// TIA Portal project "Sorting_Station" (V17)

(* hardware
DEVICE "S7-1200 station_1"  S7-1200 Station
   slot 0: "Rack_0"  S7-1200 Rack  Rack  V1.0
   slot 1: "PLC_1"  CPU 1214C DC/DC/DC  6ES7 214-1AG40-0XB0  V4.5
   slot 2: "DI 8/DQ 8x24VDC_1"  SM 1223 DI8/DQ8 x 24VDC  6ES7 223-1BH30-0XB0  V1.0
   slot 3: "AQ 2x14BIT_1"  SM 1232 AQ2  6ES7 232-4HB32-0XB0  V2.1
DEVICE "HMI_1"  KTP700 Basic PN
   slot 0: "HMI_1"  KTP700 Basic PN  6AV2 123-2GB03-0AX0  17.0.0.0
   slot 1: "HMI_RT_1"  KTP700 Basic PN  6AV2 123-2GB03-0AX0  17.0.0.0
   slot 5: "HMI_1.IE_CP_1"  PROFINET Interface  17.0.0.0
      slot 1: "PROFINET Interface_1"  PROFINET Interface
         slot 1: "Port_1"  Port
*)

// ===== PLC "PLC_1"  CPU 1214C DC/DC/DC =====

VAR_GLOBAL   // PLC tag table "Default tag table"
   "Memory_StartPB_HMI" AT %M0.0 : Bool;
END_VAR

VAR_GLOBAL   // PLC tag table "Tag_table_sorting_station"
   "I -A1" AT %I0.0 : Bool;   // Return signal E-Stop OK
   "I -K0" AT %I0.1 : Bool;   // main switch ON
   "I -S1" AT %I0.3 : Bool;   // PB Auto start
   "I -S2" AT %I0.4 : Bool;   // PB Auto Stop(in initial state)
   "I -B1" AT %I0.5 : Bool;   // Sensor cylinder M4 Retracted
   "I -B2" AT %I0.6 : Bool;   // Sensor Cylinder M4 Extented
   "I -B3" AT %I0.7 : Bool;   // Sensor motor M1 Active
   "I -B4" AT %I1.0 : Bool;   // Sensor at chute Occupied
   "I -B5" AT %I1.1 : Bool;   // Sensor metal part
   "I -B6" AT %I1.2 : Bool;   // Sensor part in front of cylinder M4
   "I -B7" AT %I1.3 : Bool;   // Sensor at End of conveyor
   "I -S3" AT %I1.4 : Bool;   // PB conveyor manual mode-Forward
   "I -S4" AT %I1.5 : Bool;   // PB conveyor manual mode-Reverse
   "I -S5" AT %I1.6 : Bool;   // PB manaul mode cylinder M4 retracts
   "I -S6" AT %I1.7 : Bool;   // PB manual mode cylinder M4 extends
   "I -S0" AT %I0.2 : Bool;   // mode selector- manual(0)/Auto(1)
   "Q -Q1" AT %Q0.0 : Bool;   // Conveyor motor M1 forward - fix speed
   "Q -Q2" AT %Q0.1 : Bool;   // Conveyor motor M1 reverse - fix speed
   "Q -Q3" AT %Q0.2 : Bool;   // Conveyor motor M1 - Variable Speed
   "Q -M2" AT %Q0.3 : Bool;   // Cylinder M4 retracts
   "Q -M3" AT %Q0.4 : Bool;   // Cylinder M4 extends
   "Q -P1" AT %Q0.5 : Bool;   // Display- main switch ON
   "Q -P2" AT %Q0.6 : Bool;   // Display- Manual mode
   "Q -P3" AT %Q0.7 : Bool;   // Display- auto mode
   "Q -P4" AT %Q1.0 : Bool;   // Display- Emergency stop activated
   "Q -P5" AT %Q1.1 : Bool;   // Display- Auto mode started
   "Q -P6" AT %Q1.2 : Bool;   // Display- Cylinder M4 Retracted
   "Q -P7" AT %Q1.3 : Bool;   // Display- Cylinder M4 Extended
   "AI -B8" AT %IW64 : Word;   // Sensor Actual value speed of motor +\- 10V
   "AI -B9" AT %IW66 : Word;   // Set point Specification via Potentiometer +\-10V
   "AO -U1" AT %QW64 : Word;   // Manipulated value speed of motor in 2 direction +\-10V
   "Temp-store-speed" AT %MW25 : Word;   // used to store 16 bit value
END_VAR

DATA_BLOCK "Motor_Auto"   // DB1
{ S7_Optimized_Access := 'FALSE' }
VERSION : 0.1
// stored: InstanceOfName Motor_Auto_mode
"Motor_Auto_mode"
BEGIN
   Setpoint_plastic_count := 5;
END_DATA_BLOCK

DATA_BLOCK "SPEED_MOTOR"   // DB2
{ S7_Optimized_Access := 'TRUE' }
VERSION : 0.1
   VAR
      Speed_Setpoint_Auto : Real := 15.0;
      Speed_Actual_Value : Real := 15.0;
      Positive_Speed : Struct   // Parameters for error/ warning positive speed
         Threshold_error : Real := 15.0;   // Speed Limit / if exceeded an error is displayed
         Threshold_Warning : Real := 10.0;   // Speed Limit / if exceeded an warning is displayed
         Error : Bool := FALSE;   // Error limit exceeded
         Warning : Bool := TRUE;   // Warning limit exceeded
      END_STRUCT;
      Negative_Speed : Struct
         Threshold_error : Real := -16.0;   // Speed Limit / if exceeded an error is displayed
         Threshold_Warning : Real := -10.0;   // Speed Limit / if exceeded an warning is displayed
         Error : Bool := FALSE;   // Error limit exceeded
         Warning : Bool := FALSE;   // Warning limit exceeded
      END_STRUCT;
      speed_setpoint_manual : Real := 5.0;
   END_VAR
BEGIN
END_DATA_BLOCK

DATA_BLOCK "MAGAZINE_PLASTIC"   // DB3
{ S7_Optimized_Access := 'TRUE' }
VERSION : 0.1
   VAR
      Setpoint_plastic_count : Int := 5;
      Actual_plastic_count : Int;
      Reset_plastic_count : Bool;
   END_VAR
BEGIN
END_DATA_BLOCK

DATA_BLOCK "OPERATING_HMI"   // DB4
{ S7_Optimized_Access := 'TRUE' }
VERSION : 0.1
   VAR
      mode_selector : Bool := false;
      automatic_start : Bool;
      automatic_stop : Bool := true;
      reset_counter_plastic : Bool;
      "Alarm Group signals01" : Word;
      "Alarm Ack Group Signals01" : Word;
   END_VAR
BEGIN
END_DATA_BLOCK

FUNCTION_BLOCK "Motor_Auto_mode"   // FB1, FBD
{ S7_Optimized_Access := 'FALSE' }
VERSION : 0.1
// The Memory_automatic_start_stop is latched with Start but only if the reset conditions are not
//  present.
//  
//  The Memory_automatic_start_stop is reset if Stop is present or safety shutoff is active or
//  automatic mode is not activated (manual mode).
//  The Conveyor_motor_automatic_mode output is activated when Memory_automatic_start_stop is
//  set, the enable conditions are met and Memory_conveyor_start_stop is set.
//  To save energy, the conveyor should only run when a part is present.
//  For this reason, the Memory_conveyor_start_stop is set when Sensor_chute_occupied signals a
//  part and reset when Sensor_end_of_conveyor produces a negative edge or safety shutoff is
//  active or automatic mode is not activated (manual mode).
// 
//  Because the Sensor_end_of_conveyor is not able to be mounted directly at the end of the
//  conveyor, the Sensor_end_of_conveyor signal must be stretched.
//  To achieve this, a latching pulse will be inserted between Sensor_end_of_conveyor and the
//  negative edge detection.
   VAR_INPUT
      Automatic_mode_active : Bool;   // Automatic mode activated
      Start : Bool;   // Pushbutton Auto start
      Stop : Bool;   // Pushbutton Auto Stop
      Enable_ok : Bool;   // All enable condition OK
      Sensor_chute_occupied : Bool;   // Sensor at chute occupied
      Safety_shutoff_active : Bool;   // Safety shutoff active e.g. Estop
      Sensor_EndofConveyor : Bool;   // Sensor part at end of conveyor
      Setpoint_plastic_count : Int;
      Reset_Counter_Workpieces_Plastic : Bool;
   END_VAR
   VAR_OUTPUT
      Conveyor_motor_auto_mode : Bool;   // Control of Conveyor motor in Auto mode
      Actual_plastic_count : Int;
   END_VAR
   VAR
      Memory_Automatic_Start_Stop : Bool;   // Memory used for start/stop automatic mode
      Memory_conveyor_start_stop : Bool;
      Memory_Edge_detection : Bool;
      IEC_Timer_Overrun : TP_TIME;
      IEC_Counter_Overrun : CTU_INT;
   END_VAR
   VAR_TEMP   // added for the SCL form of the ladder/FBD networks
      _w1 : Bool;
   END_VAR
BEGIN

REGION Network 1: Counting plastic pieces
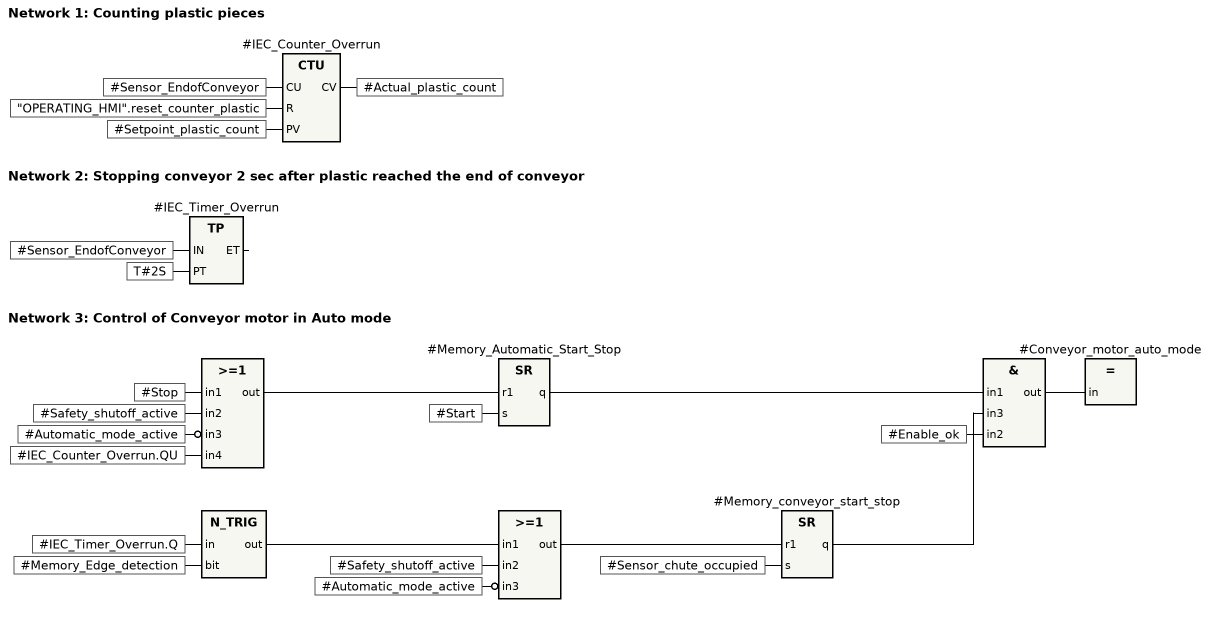
   #IEC_Counter_Overrun(CU := #Sensor_EndofConveyor,   // CTU
                        R := "OPERATING_HMI".reset_counter_plastic,
                        PV := #Setpoint_plastic_count,
                        CV => #Actual_plastic_count);
END_REGION

REGION Network 2: Stopping conveyor 2 sec after plastic reached the end of conveyor
   #IEC_Timer_Overrun(IN := #Sensor_EndofConveyor, PT := T#2S);   // TP
END_REGION

REGION Network 3: Control of Conveyor motor in Auto mode
   IF #Start THEN
       #Memory_Automatic_Start_Stop := TRUE;   // SR flip-flop
   END_IF;
   IF #Stop OR #Safety_shutoff_active OR NOT #Automatic_mode_active OR #IEC_Counter_Overrun.QU THEN
       #Memory_Automatic_Start_Stop := FALSE;
   END_IF;
   #_w1 := NOT #IEC_Timer_Overrun.Q AND #Memory_Edge_detection;   // falling edge
   #Memory_Edge_detection := #IEC_Timer_Overrun.Q;
   IF #Sensor_chute_occupied THEN
       #Memory_conveyor_start_stop := TRUE;   // SR flip-flop
   END_IF;
   IF #_w1 OR #Safety_shutoff_active OR NOT #Automatic_mode_active THEN
       #Memory_conveyor_start_stop := FALSE;
   END_IF;
   #Conveyor_motor_auto_mode := #Memory_Automatic_Start_Stop AND #Memory_conveyor_start_stop AND #Enable_ok;
END_REGION
END_FUNCTION_BLOCK

FUNCTION "Motor_manual_Mode" : Void   // FC1, FBD
TITLE = Motor control in manual mode
{ S7_Optimized_Access := 'TRUE' }
VERSION : 0.1
// conveyor motor in manual mode: If the pushbutton_manual_mode is opeerated, the enable conditions are granted and the safety shutoff is not activated the output
// Conveyor_motor_manual_mode is activated.
   VAR_INPUT
      Manual_mode_active : Bool;   // Manual mode activated
      Pushbutton_manual_mode : Bool;   // Pushbutton manual mode conveyor on
      Enable_OK : Bool;   // All enable conditions OK
      Safety_shutoff_active : Bool;   // Saftey shutoff active
      Forward_signal : Bool;   // signal for operation in forward direction
      Backward_signal : Bool;   // signal for operation in reverse direction
      manual_motor_speed : Real;   // speed of motor for manual mode in either direction
   END_VAR
   VAR_OUTPUT
      Conveyor_mode_manual_mode : Bool;   // Control of the conveyor motor in manual mode
      Output_motor_speed : Real;   // speed of motor in manual mode
   END_VAR
   VAR_TEMP
      negative_value : Real;
      "Speed*2" : Real;
   END_VAR
BEGIN

REGION Network 1: Control of the conveyor in manual mode.
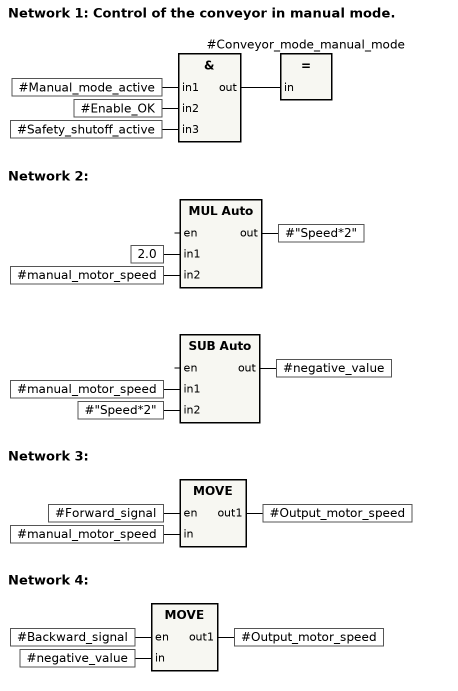
   #Conveyor_mode_manual_mode := #Manual_mode_active AND #Enable_OK AND #Safety_shutoff_active;
END_REGION

REGION Network 2
   #"Speed*2" := 2.0 * #manual_motor_speed;
   #negative_value := #manual_motor_speed - #"Speed*2";
END_REGION

REGION Network 3
   IF #Forward_signal THEN #Output_motor_speed := #manual_motor_speed; END_IF;
END_REGION

REGION Network 4
   IF #Backward_signal THEN #Output_motor_speed := #negative_value; END_IF;
END_REGION
END_FUNCTION

FUNCTION "Copy 16bit data" : Void   // FC2, SCL
{ S7_Optimized_Access := 'TRUE' }
VERSION : 0.1
   VAR_INPUT
      "Copy speed from" : Int;
   END_VAR
   VAR_OUTPUT
      "Copy speed to" : Int;
   END_VAR
BEGIN
   #"Copy speed to" := #"Copy speed from";
END_FUNCTION

FUNCTION "Assign_discrete_alarms" : Void   // FC3, FBD
{ S7_Optimized_Access := 'TRUE' }
VERSION : 0.1
   VAR_INPUT
      discrete_alarm_X0 : Bool;
      discrete_alarm_X1 : Bool;
      discrete_alarm_X2 : Bool;
      discrete_alarm_X3 : Bool;
   END_VAR
   VAR_OUTPUT
      group_signal01 : Word;
   END_VAR
BEGIN

REGION Network 1
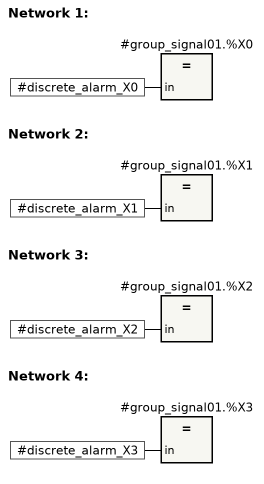
   #group_signal01.%X0 := #discrete_alarm_X0;
END_REGION

REGION Network 2
   #group_signal01.%X1 := #discrete_alarm_X1;
END_REGION

REGION Network 3
   #group_signal01.%X2 := #discrete_alarm_X2;
END_REGION

REGION Network 4
   #group_signal01.%X3 := #discrete_alarm_X3;
END_REGION
END_FUNCTION

FUNCTION "MOTOR_SPEEDMONITORING" : Void   // FC11, FBD
{ S7_Optimized_Access := 'TRUE' }
VERSION : 0.1
// In the "MOTOR_SPEED_MONITORING" [FC11] function, the actual value is made available at 
// B8 as an analog value and is queried at an input of the "MOTOR_SPEEDMONITORING" [FC11]
//  function.
//  The actual speed value is scaled to revolutions per minute (range: +/- 50 rpm) and made
//  available at an output.
//  The following four limits can be specified at the block inputs in order to monitor them in the
//  function:
//  Speed > Speed limit error max
//  Speed > Speed limit warning max
//  Speed  < Speed limit warning min
//  Speed  < Speed limit warning min
//  If a limit is exceeded or undershot, the value TRUE (1) is assigned to the corresponding output
//  bit.
//  If a fault is present, the safety shutoff of the "MOTOR_AUTO" [FB1] function block is to be
//  triggered
   VAR_INPUT
      Actual_Speed_AI : Int;
      Speed_limit_error_max : Real;
      Speed_limit_warning_max : Real;
      Speed_limit_warning_min : Real;
      Speed_limit_error_min : Real;
   END_VAR
   VAR_OUTPUT
      Speed_warning_max : Bool;
      Speed_warning_min : Bool;
      Speed_error_max : Bool;
      Speed_error_min : Bool;
      Motor_speed_AO : Real;
   END_VAR
   VAR_TEMP
      Motor_speed_Norm : Real;
      Actual_speed_Scaled : Real;
   END_VAR
BEGIN

REGION Network 1: Normalisation
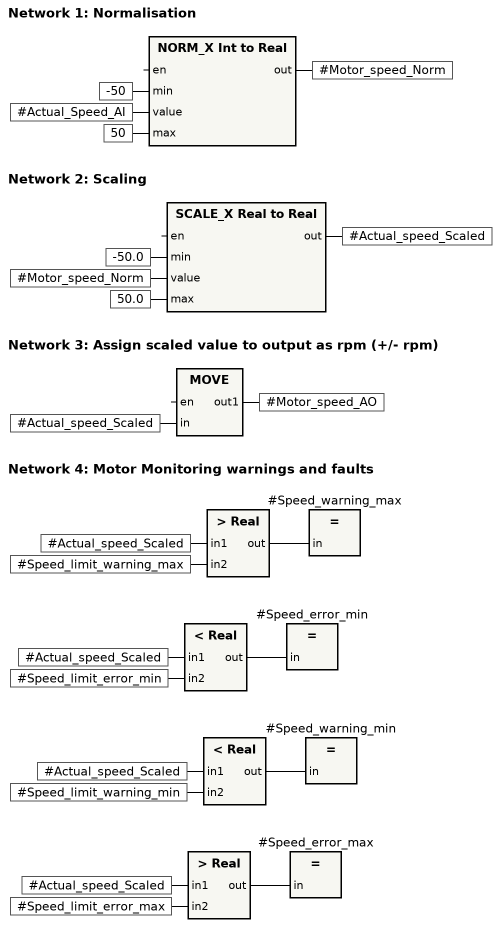
   #Motor_speed_Norm := NORM_X(MIN := -50, VALUE := #Actual_Speed_AI, MAX := 50);
END_REGION

REGION Network 2: Scaling
   #Actual_speed_Scaled := SCALE_X(MIN := -50.0, VALUE := #Motor_speed_Norm, MAX := 50.0);
END_REGION

REGION Network 3: Assign scaled value to output as rpm (+/- rpm)
   #Motor_speed_AO := #Actual_speed_Scaled;
END_REGION

REGION Network 4: Motor Monitoring warnings and faults
   #Speed_warning_max := #Actual_speed_Scaled > #Speed_limit_warning_max;
   #Speed_error_min := #Actual_speed_Scaled < #Speed_limit_error_min;
   #Speed_warning_min := #Actual_speed_Scaled < #Speed_limit_warning_min;
   #Speed_error_max := #Actual_speed_Scaled > #Speed_limit_error_max;
END_REGION
END_FUNCTION

ORGANIZATION_BLOCK "Main"   // OB1, FBD, ProgramCycle
TITLE = "Main Program Sweep (Cycle)"
{ S7_Optimized_Access := 'TRUE' }
VERSION : 0.1
// The "MOTOR_AUTO" [FB1] function block controls a conveyor in automatic mode.
//  The Memory_Automatic_Start_Stop is switched on in a latching manner with Start, but only if the
//  reset conditions are not present.
//  The Memory_Automatic_Start_Stop is to be reset if Stop is pending, the safety shutoff is active
//  or automatic mode is not activated from the visualization.
//  The Automatic_Motor output is controlled when Memory_Automatic_Start_Stop is set, the
//  enabling conditions are met and Memory_Conveyor_Start_Stop is set.
//  For energy saving reasons, the conveyor is to run only when a transport part is present.
//  Therefore, Memory_Conveyor_Start_Stop is set if Sensor_slide signals a part and is reset if
//  Sensor_end_of_conveyor generates a negative edge or the safety shutoff is active or automatic
//  mode is not activated (manual mode).
//  Because Sensor_end_of_conveyor is not mounted directly at the end of the conveyor, a signal
//  delay of the Sensor_end_of_conveyor signal is programmed.
//  The magazine for plastics holds only five parts. Therefore, the parts are counted at the end of
//  the conveyor. If the magazine contains five parts, automatic mode is to be stopped. After the
//  magazine is emptied, automatic mode is restarted with another Start, once the counter has been
//  reset from the visualization.
//  The speed is specified with an input in the "MOTOR_SPEEDCONTROL" [FC10] function in
//  revolutions per minute (range: +/- 50 rpm).
//  The speed setpoint is first checked in the function for correct input in the range +/- 50 rpm.
//  If the speed setpoint is outside the range +/- 50 rpm, the value 0 is output at the speed setpoint
//  output. The value TRUE (1) is assigned to the return value of the function (Ret_Val).
//  If the specified speed is in the range +/- 50 rpm, this value is first scaled to the range 0…1 and
//  then scaled for the output as manipulated speed value at the analog output to +/- 27648 with
//  data type 16-bit integer (Int).
//  In the "MOTOR_SPEED_MONITORING" [FC11] function, the actual value is made available at 
// B8 as an analog value and is queried at an input of the "MOTOR_SPEEDMONITORING" [FC11]
//  function.
//  The actual speed value is scaled to revolutions per minute (range: +/- 50 rpm) and made
//  available at an output.
//  The following four limits can be specified at the block inputs in order to monitor them in the
//  function:
//  Speed > Speed limit error max
//  Speed > Speed limit warning max
//  Speed  < Speed limit warning min
//  Speed  < Speed limit warning min
//  If a limit is exceeded or undershot, the value TRUE (1) is assigned to the corresponding output
//  bit.
//  If a fault is present, the safety shutoff of the "MOTOR_AUTO" [FB1] function block is to be
//  triggered.
//  Speed setpoint and actual speed value as well as the positive and negative error and warning
//  limits are created in the "SPEED_MOTOR" [DB2] data block, as are the error and warning bits.
//  The setpoint and actual value of the counter for plastic parts will be specified and displayed in
//  the global "MAGAZINE_PLASTIC" [DB3] data block. These values are connected with the
//  "MOTOR_AUTO" [FB1] function block via an input for specification of the setpoint and via an
//  output for display of the actual value
   VAR_INPUT
      Initial_Call : Bool;   // Initial call of this OB
      Remanence : Bool;   // =True, if remanent data are available
   END_VAR
BEGIN

REGION Network 1: Delete this block if you have real motor connected and actual feedback from field
   // Modify MW25 to read Motor speed value in HMI
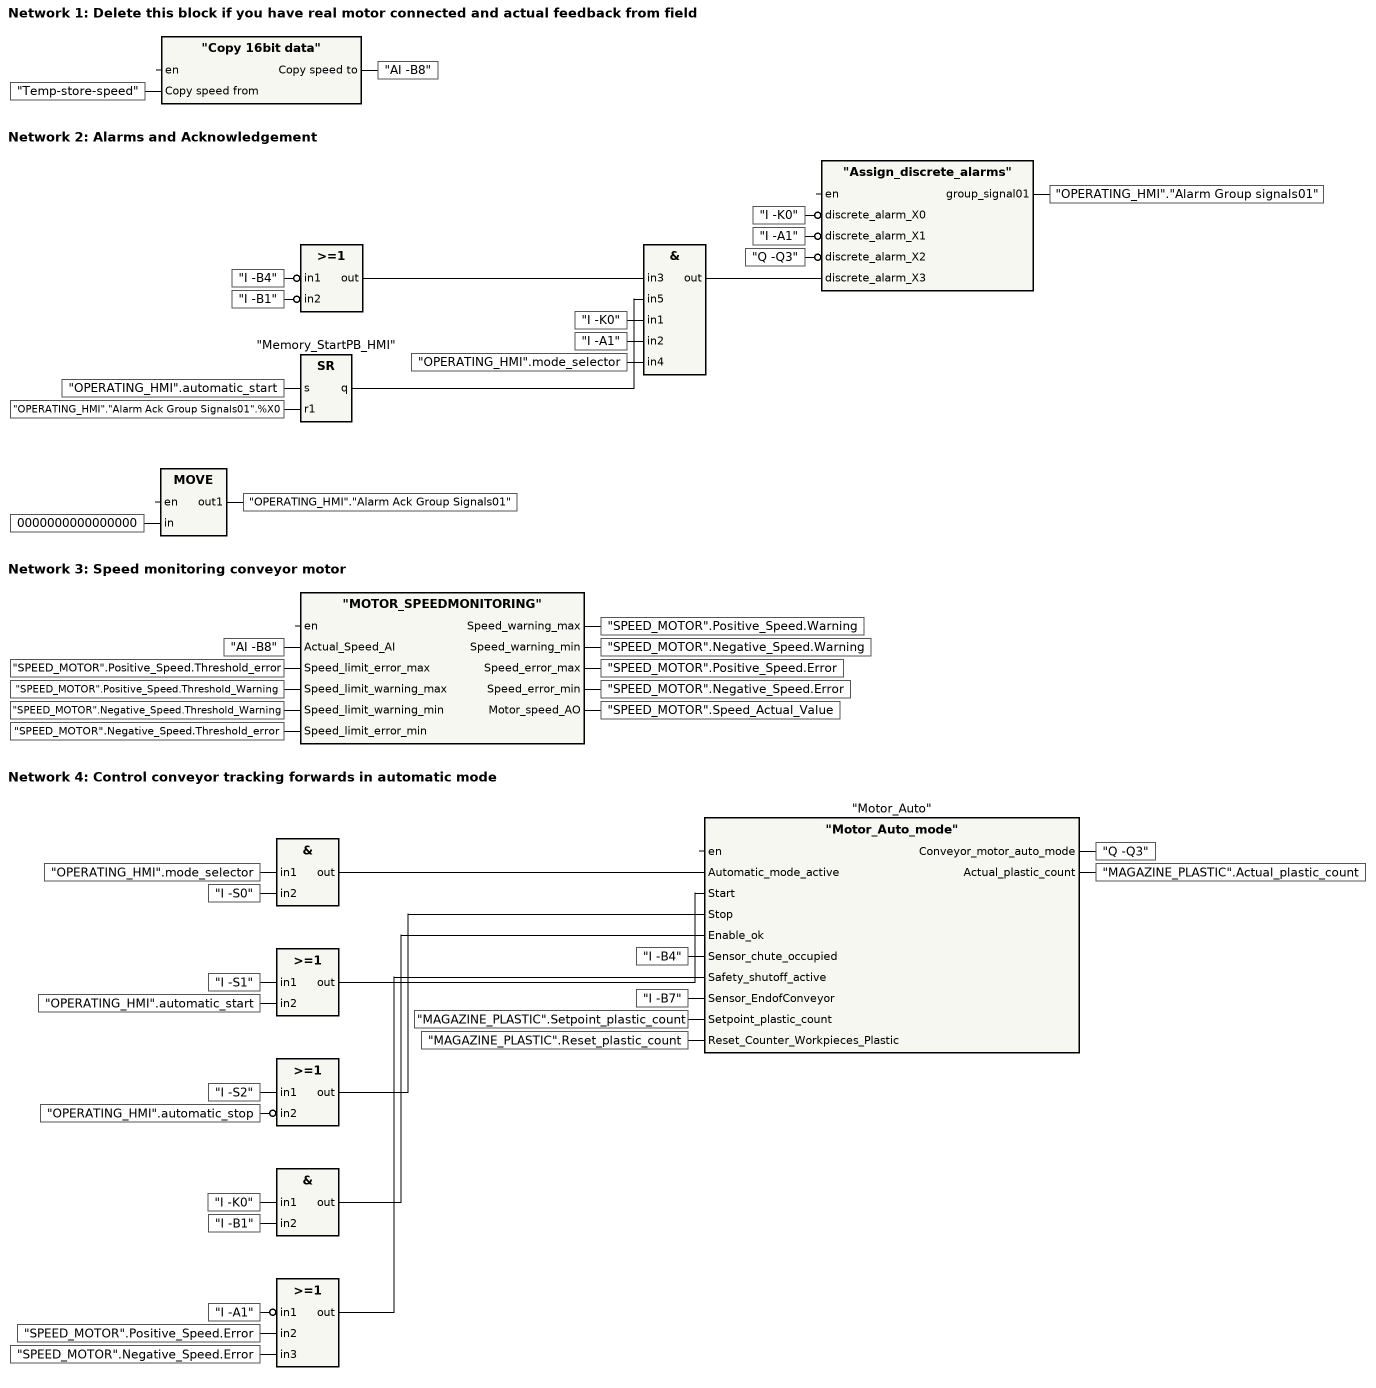
   "Copy 16bit data"("Copy speed from" := "Temp-store-speed", "Copy speed to" => "AI -B8");
END_REGION

REGION Network 2: Alarms and Acknowledgement
   IF "OPERATING_HMI".automatic_start THEN
       "Memory_StartPB_HMI" := TRUE;   // SR flip-flop
   END_IF;
   IF "OPERATING_HMI"."Alarm Ack Group Signals01".%X0 THEN "Memory_StartPB_HMI" := FALSE; END_IF;
   "Assign_discrete_alarms"(discrete_alarm_X0 := NOT "I -K0",
                           discrete_alarm_X1 := NOT "I -A1",
                           discrete_alarm_X2 := NOT "Q -Q3",
                           discrete_alarm_X3 := (NOT "I -B4" OR NOT "I -B1") AND "Memory_StartPB_HMI" AND "I -K0" AND "I -A1" AND "OPERATING_HMI".mode_selector,
                           group_signal01 => "OPERATING_HMI"."Alarm Group signals01");
   "OPERATING_HMI"."Alarm Ack Group Signals01" := 0000000000000000;
END_REGION

REGION Network 3: Speed monitoring conveyor motor
   "MOTOR_SPEEDMONITORING"(Actual_Speed_AI := "AI -B8",
                           Speed_limit_error_max := "SPEED_MOTOR".Positive_Speed.Threshold_error,
                           Speed_limit_warning_max := "SPEED_MOTOR".Positive_Speed.Threshold_Warning,
                           Speed_limit_warning_min := "SPEED_MOTOR".Negative_Speed.Threshold_Warning,
                           Speed_limit_error_min := "SPEED_MOTOR".Negative_Speed.Threshold_error,
                           Speed_warning_max => "SPEED_MOTOR".Positive_Speed.Warning,
                           Speed_warning_min => "SPEED_MOTOR".Negative_Speed.Warning,
                           Speed_error_max => "SPEED_MOTOR".Positive_Speed.Error,
                           Speed_error_min => "SPEED_MOTOR".Negative_Speed.Error,
                           Motor_speed_AO => "SPEED_MOTOR".Speed_Actual_Value);
END_REGION

REGION Network 4: Control conveyor tracking forwards in automatic mode
   "Motor_Auto"(Automatic_mode_active := "OPERATING_HMI".mode_selector AND "I -S0",   // "Motor_Auto_mode"
                Start := "I -S1" OR "OPERATING_HMI".automatic_start,
                Stop := "I -S2" OR NOT "OPERATING_HMI".automatic_stop,
                Enable_ok := "I -K0" AND "I -B1",
                Sensor_chute_occupied := "I -B4",
                Safety_shutoff_active := NOT "I -A1" OR "SPEED_MOTOR".Positive_Speed.Error OR "SPEED_MOTOR".Negative_Speed.Error,
                Sensor_EndofConveyor := "I -B7",
                Setpoint_plastic_count := "MAGAZINE_PLASTIC".Setpoint_plastic_count,
                Reset_Counter_Workpieces_Plastic := "MAGAZINE_PLASTIC".Reset_plastic_count,
                Conveyor_motor_auto_mode => "Q -Q3",
                Actual_plastic_count => "MAGAZINE_PLASTIC".Actual_plastic_count);
END_REGION

REGION Network 5: Control conveyor motor forwards in manual mode
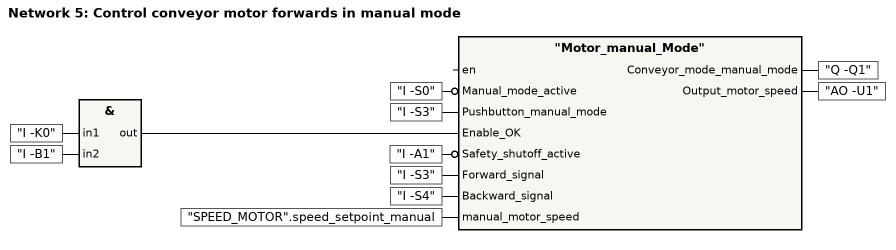
   "Motor_manual_Mode"(Manual_mode_active := NOT "I -S0",
                       Pushbutton_manual_mode := "I -S3",
                       Enable_OK := "I -K0" AND "I -B1",
                       Safety_shutoff_active := NOT "I -A1",
                       Forward_signal := "I -S3",
                       Backward_signal := "I -S4",
                       manual_motor_speed := "SPEED_MOTOR".speed_setpoint_manual,
                       Conveyor_mode_manual_mode => "Q -Q1",
                       Output_motor_speed => "AO -U1");
END_REGION
END_ORGANIZATION_BLOCK

ORGANIZATION_BLOCK "Cyclic interrupt"   // OB30, FBD, CyclicInterrupt
{ S7_Optimized_Access := 'TRUE' }
VERSION : 0.1
   VAR_INPUT
      Initial_Call : Bool;   // Initial call of this OB
      Event_Count : Int;   // Events discarded
   END_VAR
BEGIN

REGION Network 1
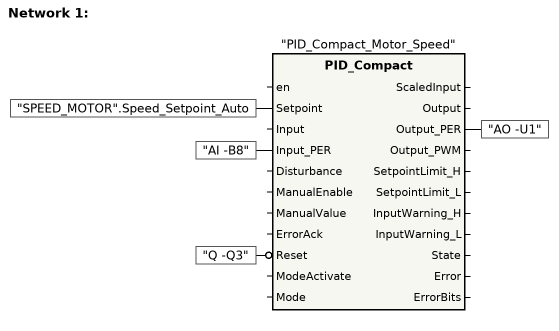
   "PID_Compact_Motor_Speed"(Setpoint := "SPEED_MOTOR".Speed_Setpoint_Auto,   // PID_Compact
                           Input_PER := "AI -B8",
                           Reset := NOT "Q -Q3",
                           Output_PER => "AO -U1");
END_REGION
END_ORGANIZATION_BLOCK

(* ===== HMI "HMI_RT_1" =====
system functions are stored by id; their names below are inferred from use
connection "HMI_Connection_1": ETHERNET, SMART_S7_1200_OMS

HMI tags "Default tag table"
   "Tag_ScreenNumber" : UInt, internal
   "SPEED_MOTOR_Speed_Actual_Value" : Real = PLC SPEED_MOTOR.Speed_Actual_Value, 100 ms
   "I -B4" : Bool = PLC "I -B4" AT %I1.0, 100 ms
   "I -B5" : Bool = PLC "I -B5" AT %I1.1, 100 ms
   "I -B6" : Bool = PLC "I -B6" AT %I1.2, 100 ms
   "I -B7" : Bool = PLC "I -B7" AT %I1.3, 100 ms
   "I -B2" : Bool = PLC "I -B2" AT %I0.6, 100 ms
   "I -B1" : Bool = PLC "I -B1" AT %I0.5, 100 ms
   "I -B3" : Bool = PLC "I -B3" AT %I0.7, 100 ms
   "Q -Q3" : Bool = PLC "Q -Q3" AT %Q0.2, 100 ms
   "OPERATING_HMI_reset_counter_plastic" : Bool = PLC OPERATING_HMI.reset_counter_plastic, 100 ms
   "MAGAZINE_PLASTIC_Actual_plastic_count" : Int = PLC MAGAZINE_PLASTIC.Actual_plastic_count, 100 ms
   "OPERATING_HMI_automatic_start" : Bool = PLC OPERATING_HMI.automatic_start, 100 ms
   "OPERATING_HMI_automatic_stop" : Bool = PLC OPERATING_HMI.automatic_stop, 100 ms
   "I -A1" : Bool = PLC "I -A1" AT %I0.0, 100 ms
   "I -K0" : Bool = PLC "I -K0" AT %I0.1, 100 ms
   "Motor_Auto_Memory_Automatic_Start_Stop" : Bool = PLC Motor_Auto.Memory_Automatic_Start_Stop AT %DB1.DBX10.0, 100 ms
   "SPEED_MOTOR_Speed_Setpoint" : Real = PLC SPEED_MOTOR.Speed_Setpoint_Auto, 100 ms
   "SPEED_MOTOR_Positive_Speed_Threshold_error" : Real = PLC SPEED_MOTOR.Positive_Speed.Threshold_error, 100 ms
   "SPEED_MOTOR_Positive_Speed_Threshold_Warning" : Real = PLC SPEED_MOTOR.Positive_Speed.Threshold_Warning, 100 ms
   "SPEED_MOTOR_Negative_Speed_Threshold_error" : Real = PLC SPEED_MOTOR.Negative_Speed.Threshold_error, 100 ms
   "SPEED_MOTOR_Negative_Speed_Threshold_Warning" : Real = PLC SPEED_MOTOR.Negative_Speed.Threshold_Warning, 100 ms
   "OPERATING_HMI_Group signals01" : Word = PLC OPERATING_HMI."Alarm Group signals01", 1 s
   "MAGAZINE_PLASTIC_Setpoint_plastic_count" : Int = PLC MAGAZINE_PLASTIC.Setpoint_plastic_count, 1 s
   "SPEED_MOTOR_Positive_Speed_Error" : Bool = PLC SPEED_MOTOR.Positive_Speed.Error, 1 s
   "SPEED_MOTOR_Positive_Speed_Warning" : Bool = PLC SPEED_MOTOR.Positive_Speed.Warning, 1 s
   "SPEED_MOTOR_Negative_Speed_Warning" : Bool = PLC SPEED_MOTOR.Negative_Speed.Warning, 1 s
   "SPEED_MOTOR_Negative_Speed_Error" : Bool = PLC SPEED_MOTOR.Negative_Speed.Error, 1 s
   "Motor_Auto_Setpoint_plastic_count" : Int = PLC Motor_Auto.Setpoint_plastic_count AT %DB1.DBW2, 1 s
   "OPERATING_HMI_mode_selector" : Bool = PLC OPERATING_HMI.mode_selector, 1 s
   "SPEED_MOTOR_speed_setpoint_manual" : Real = PLC SPEED_MOTOR.speed_setpoint_manual, 1 s
   "OPERATING_HMI_Alarm Ack Group Signals01" : Word = PLC OPERATING_HMI."Alarm Ack Group Signals01", 1 s

discrete alarms
   1: 'Main switch OFF', class Warnings, trigger "OPERATING_HMI_Group signals01" bit 0
   2: 'Auto Mode OFF', class Warnings, trigger "OPERATING_HMI_Group signals01" bit 2
   3: 'Emergency Activated!', class Warnings, trigger "OPERATING_HMI_Group signals01" bit 1
   4: 'Check if B4 sensor has detected an item or if M4 cylinder is retracted.', class Acknowledgement, trigger "OPERATING_HMI_Group signals01" bit 3

analog alarms
   1: 'Error threshold exceeded motor pos. speed', class Errors, trigger "SPEED_MOTOR_Speed_Actual_Value"
   2: 'Warning threshold exceeded motor pos. speed', class Warnings, trigger "SPEED_MOTOR_Speed_Actual_Value"
   3: 'Error threshold underran motor pos. speed', class Errors, trigger "SPEED_MOTOR_Speed_Actual_Value"
   4: 'Warning threshold underran motor pos. speed', class Warnings, trigger "SPEED_MOTOR_Speed_Actual_Value"

text list "Text_list_emergency_stop": 0 'Emergency Stop released'; 1 'Emergency Stop OK'

text list "Text_list_main_switch": 0 'main switch OFF'; 1 'main switch ON'

text list "Text_list_automatic": 0 'automatic stopped'; 1 'automatic started'

text list "Text_list_plastic_count_setpoint": 1 '1'; 2 '2'; 3 '3'; 4 '4'; 5 '5'; 6 '6'; 7 '7'; 8 '8'; 9 '9'; 10 '10'; 11 '11'; 12 '12'; 13 '13'; 14 '14'; 15 '15'; 16 '16'; 17 '17'; 18 '18'; 19 '19'; 20 '20'

text list "Text_list_Motor_manual_speed": 1 '1'; 2 '2'; 3 '3'; 4 '4'; 6 '6'; 7 '7'; 8 '8'; 9 '9'; 10 '10'; 5 '5'

graphic list "Graphic_list_warning": 0 'Warning'; 1 'Logo of HMI_1'

Template "Template_1" 800x480
   Button "Exit" at 714,429 size 71x50; TextOff 'Exit'; PictureOff "ExitRuntime_KTP700_Basic_PN_TR"; PictureOn "ExitRuntime_KTP700_Basic_PN_TR"
      on Release: StopRuntime(0)
   Button "Template_Button" at 614,429 size 71x50; TextOff 'Text'
   Button "Template_Button_1" at 514,429 size 71x50; TextOff 'Text'
   Button "Template_Button_2" at 414,429 size 71x50; TextOff 'Text'
   Button "Template_Button_3" at 314,429 size 71x50; TextOff 'Text'; PictureOff "Navigates to User administration for KTP700 Basic+ PN 17.0.0.0"
      on Release: ActivateScreen("User administration", 0)
   Button "Template_Button_4" at 214,429 size 71x50; TextOff 'Text'; PictureOff "Navigates to System screens for KTP700 Basic+ PN 17.0.0.0"
      on Release: ActivateScreen("System screens", 0)
   Button "Alarms" at 114,429 size 71x50; TextOff 'Alarms'; PictureOff "AlarmDisplay_KTP700_Basic_PN_TR"; PictureOn "AlarmDisplay_KTP700_Basic_PN_TR"
      on Release: function_ef3f5d25("Alarm window_Unacknowledged", -1)
   Button "Start screen" at 14,429 size 71x50; TextOff 'Start screen'; PictureOff "NavigateHome_KTP700_Basic_PN_TR"; PictureOn "NavigateHome_KTP700_Basic_PN_TR"
      on Release: ActivateScreen("Overview Sorting_station", 0)
   SymbolicIOField "Symbolic_IO_Field_Screen" at 254,8 size 268x33; TextOff '0'; TextOn '1'; TextList "TextList_ScreenNames"
      ProcessValue <- "Tag_ScreenNumber"
      on Change: ActivateScreenByNumber("Tag_ScreenNumber", 0)
   DateTimeField "HmiScreenItemData" at 695,25 size 105x25
   DateTimeField "HmiScreenItemData_1" at 695,0 size 105x25
   GraphicIOField "Template_Graphic I/O field_1" at 0,0 size 50x50; PictureList "Graphic_list_warning"
      ProcessValue <- "I -A1"
   SymbolicIOField "Template_Symbolic I/O field_1" at 50,9 size 201x32; TextOff '0'; TextOn '1'; TextList "Text_list_emergency_stop"
      ProcessValue <- "I -A1"
   SymbolicIOField "Template_Symbolic I/O field_2" at 525,1 size 167x26; TextOn '1'; TextOff '0'; TextList "Text_list_main_switch"
      ProcessValue <- "I -K0"
      Appearance <- "I -K0"
   SymbolicIOField "Template_Symbolic I/O field_3" at 525,25 size 167x27; TextOn '1'; TextOff '0'; TextList "Text_list_automatic"
      ProcessValue <- "Motor_Auto_Memory_Automatic_Start_Stop"
      Appearance <- "Motor_Auto_Memory_Automatic_Start_Stop"

screen "Overview Sorting_station" 800x480, template "Template_1"
   on GenerateScreen: SetTag("Tag_ScreenNumber", 1)
   Button "HmiScreenItemData" at 31,65 size 150x47; TextOff 'Speed motor'; PictureOff "Navigates to Speed motor for KTP700 Basic+ PN 17.0.0.0"; PictureOn "Navigates to Speed motor for KTP700 Basic+ PN 17.0.0.0"
      on Release: ActivateScreen("Speed motor", 0)
   Button "HmiScreenItemData_1" at 194,65 size 150x47; TextOff 'Magazine plastic'; PictureOff "Navigates to Magazine plastic for KTP700 Basic+ PN 17.0.0.0"; PictureOn "Navigates to Magazine plastic for KTP700 Basic+ PN 17.0.0.0"
      on Release: ActivateScreen("Magazine plastic", 0)
   GraphicView "Graphic view_1" at 16,130 size 765x268; Picture "conveyor_process_image"
   IOField "I/O field_1" at 194,347 size 80x33; FormatPattern s999.99
      ProcessValue <- "SPEED_MOTOR_Speed_Actual_Value"
   TextField "Text field_1" at 31,347 size 163x23; Text 'Speed Actual Value'
   TextField "Text field_2" at 276,347 size 42x23; Text 'RPM'
   Rectangle "Rectangle_1" at 172,202 size 13x13
      Appearance <- "I -B4"
   Rectangle "Rectangle_2" at 272,202 size 13x13
      Appearance <- "I -B5"
   Rectangle "Rectangle_3" at 446,153 size 13x13
      Appearance <- "I -B6"
   Rectangle "Rectangle_4" at 702,203 size 13x13
      Appearance <- "I -B7"
   Rectangle "Rectangle_5" at 492,309 size 13x13
      Appearance <- "I -B2"
   Rectangle "Rectangle_6" at 492,367 size 13x13
      Appearance <- "I -B1"
   Rectangle "Rectangle_7" at 196,327 size 13x13
      Appearance <- "I -B3"
   TextField "Text field_3" at 54,321 size 138x23; Text 'M1 Motor Active'
   Line "Line_1" at 432,249 size 77x1
      Visibility <- "Q -Q3"
   Line "Line_2" at 196,250 size 75x0
      Visibility <- "Q -Q3"
   Button "Button_1" at 674,322 size 96x32; TextOff 'Reset'
      on Press: function_b14e0dd5("OPERATING_HMI_reset_counter_plastic", 0)
   TextField "Text field_4" at 542,298 size 225x23; Text 'Counter workpieces plastic'
   IOField "I/O field_2" at 601,322 size 66x32; FormatPattern 99
      ProcessValue <- "MAGAZINE_PLASTIC_Actual_plastic_count"
   Button "Button_2" at 605,63 size 50x50; TextOff 'Start'; PictureOff "Pushbutton-Round-G_Off_256c"; PictureOn "Pushbutton-Round-G_On_256c"
      on Press: function_b14e0dd5("OPERATING_HMI_automatic_start", 0)
   Button "Button_3" at 675,63 size 50x50; TextOff 'Stop'; PictureOff "Pushbutton-Stop_Off_256c"; PictureOn "Pushbutton-Stop_On_256c"
      on Press: ResetBit("OPERATING_HMI_automatic_stop")
      on Release: SetBit("OPERATING_HMI_automatic_stop")
   IOField "I/O field_3" at 601,363 size 66x32; FormatPattern 99
      ProcessValue <- "MAGAZINE_PLASTIC_Setpoint_plastic_count"
   TextField "Text field_5" at 544,325 size 57x23; Text 'Actual'
   TextField "Text field_6" at 546,364 size 26x23; Text 'SV'
   TextField "Text field_8" at 417,85 size 55x22; Text 'MODE:'
   TextField "Text field_7" at 380,65 size 100x22; Text 'OPERATING'
   Switch "Switch_1" at 486,63 size 101x48; CaptionText 'Switch'; TextOff 'Man'; TextOn 'Auto'
      on SwitchOn: SetBit("OPERATING_HMI_mode_selector")
      on SwitchOff: ResetBit("OPERATING_HMI_mode_selector")
      ProcessValue <- "OPERATING_HMI_mode_selector"

screen "Speed motor" 800x480, template "Template_1"
   on GenerateScreen: SetTag("Tag_ScreenNumber", 2)
   Button "Back" at 1,52 size 159x47; TextOff 'Back'
      on Release: ActivateScreen("Overview Sorting_station", 0)
   Bar "Bar_1" at 128,182 size 71x244; MinimumValue -50; MaximumValue 50
      ProcessValue <- "SPEED_MOTOR_Speed_Actual_Value"
   TextField "Text field_1" at 0,153 size 118x23; Text 'Actual Value'
   IOField "I/O field_1" at 127,108 size 72x31; FormatPattern s99.99
      ProcessValue <- "SPEED_MOTOR_Speed_Setpoint"
   TextField "Text field_2" at 42,112 size 74x23; Text 'Setpoint'
   IOField "I/O field_2" at 127,151 size 72x31; FormatPattern s99.99
      ProcessValue <- "SPEED_MOTOR_Speed_Actual_Value"
   TextField "Text field_3" at 299,65 size 108x23; Text 'Speed Motor'
   TextField "Text field_4" at 263,116 size 290x23; Text 'Error max threshold positive speed'
   TextField "Text field_5" at 264,173 size 317x23; Text 'Warning max threshold positive speed'
   TextField "Text field_6" at 262,284 size 290x23; Text 'Error max threshold positive speed'
   TextField "Text field_7" at 264,229 size 317x23; Text 'Warning max threshold positive speed'
   IOField "I/O field_3" at 602,107 size 77x32; FormatPattern 999
      ProcessValue <- "SPEED_MOTOR_Positive_Speed_Threshold_error"
   IOField "I/O field_4" at 602,164 size 77x32; FormatPattern 999
      ProcessValue <- "SPEED_MOTOR_Positive_Speed_Threshold_Warning"
   IOField "I/O field_5" at 602,275 size 77x32; FormatPattern 999
      ProcessValue <- "SPEED_MOTOR_Negative_Speed_Threshold_error"
   IOField "I/O field_6" at 602,220 size 77x32; FormatPattern 999
      ProcessValue <- "SPEED_MOTOR_Negative_Speed_Threshold_Warning"
   Ellipse "Ellipse_1" at 716,105 size 34x34
      Appearance <- "SPEED_MOTOR_Positive_Speed_Error"
   Ellipse "Ellipse_2" at 716,162 size 34x34
      Appearance <- "SPEED_MOTOR_Positive_Speed_Warning"
   Ellipse "Ellipse_3" at 716,218 size 34x34
      Appearance <- "SPEED_MOTOR_Negative_Speed_Warning"
   Ellipse "Ellipse_4" at 716,273 size 34x34
      Appearance <- "SPEED_MOTOR_Negative_Speed_Error"
   TextField "Text field_8" at 263,358 size 171x23; Text 'Motor manual speed'
   SymbolicIOField "Symbolic I/O field_1" at 446,354 size 96x32; TextOff '0'; TextOn '1'; TextList "Text_list_Motor_manual_speed"
      ProcessValue <- "SPEED_MOTOR_speed_setpoint_manual"

screen "Magazine plastic" 800x480, template "Template_1"
   on GenerateScreen: SetTag("Tag_ScreenNumber", 3)
   Button "Back" at 1,52 size 159x47; TextOff 'Back'
      on Release: ActivateScreen("Overview Sorting_station", 0)
   Button "Button_1" at 92,347 size 96x32; TextOff 'Reset'
      on Press: function_b14e0dd5("OPERATING_HMI_reset_counter_plastic", 0)
   TextField "Text field_4" at 258,54 size 225x23; Text 'Counter workpieces plastic'
   TextField "Text field_5" at 207,96 size 57x23; Text 'Actual'
   TextField "Text field_6" at 352,96 size 74x23; Text 'Setpoint'
   Bar "Bar_1" at 200,127 size 70x280; MinimumValue 0; MaximumValue 20
      ProcessValue <- "MAGAZINE_PLASTIC_Actual_plastic_count"
   IOField "I/O field_1" at 92,302 size 96x32; FormatPattern 99
      ProcessValue <- "MAGAZINE_PLASTIC_Actual_plastic_count"
   SymbolicIOField "Symbolic I/O field_1" at 350,128 size 84x32; TextOff '0'; TextOn '1'; TextList "Text_list_plastic_count_setpoint"
      ProcessValue <- "MAGAZINE_PLASTIC_Setpoint_plastic_count"

screen "System screens" 800x480, template "Template_1"
   on GenerateScreen: SetTag("Tag_ScreenNumber", 4)
   Button "Back" at 1,52 size 159x47; TextOff 'Back'
      on Release: ActivateScreen("Overview Sorting_station", 0)
   Button "HmiScreenItemData" at 286,83 size 159x47; TextOff 'SIMATIC PLC system diagnos...'; PictureOff "Navigates to SIMATIC PLC system diagnostics for KTP700 Basic+ PN 17.0.0.0"; PictureOn "Navigates to SIMATIC PLC system diagnostics for KTP700 Basic+ PN 17.0.0.0"; Authorization "User administration"
      on Release: ActivateScreen("SIMATIC PLC system diagnostics", 0)
   Button "HmiScreenItemData_1" at 287,217 size 159x47; TextOff 'Project information'; PictureOff "Navigates to Project information for KTP700 Basic+ PN 17.0.0.0"; PictureOn "Navigates to Project information for KTP700 Basic+ PN 17.0.0.0"
      on Release: ActivateScreen("Project information", 0)
   Button "HmiScreenItemData_3" at 288,282 size 159x47; TextOff 'System information'; PictureOff "Navigates to System information for KTP700 Basic+ PN 17.0.0.0"; PictureOn "Navigates to System information for KTP700 Basic+ PN 17.0.0.0"
      on Release: ActivateScreen("System information", 0)
   Button "HmiScreenItemData_4" at 287,151 size 159x47; TextOff 'Different jobs'; PictureOff "Navigates to Different jobs for KTP700 Basic+ PN 17.0.0.0"; PictureOn "Navigates to Different jobs for KTP700 Basic+ PN 17.0.0.0"; Authorization "User administration"
      on Release: ActivateScreen("Different jobs", 0)

screen "SIMATIC PLC system diagnostics" 800x480, template "Template_1"
   on GenerateScreen: SetTag("Tag_ScreenNumber", 5)
   SysDiagControl "HmiScreenItemData" at 1,100 size 796x321
   Button "Back" at 1,52 size 159x47; TextOff 'Back'
      on Release: ActivateScreen("System screens", 0)

screen "Project information" 800x480, template "Template_1"
   on GenerateScreen: SetTag("Tag_ScreenNumber", 6)
   TextField "HmiScreenItemData" at 35,102 size 171x28; Text 'Project name:'
   TextField "HmiScreenItemData_1" at 241,102 size 524x28; Text 'Sorting_Station'
   TextField "HmiScreenItemData_2" at 35,132 size 171x28; Text 'Created on:'
   TextField "HmiScreenItemData_3" at 241,132 size 524x28; Text '5/8/2025 6:37:35 AM'
   TextField "HmiScreenItemData_4" at 35,162 size 171x28; Text 'Author:'
   TextField "HmiScreenItemData_5" at 241,162 size 524x28; Text 'Aman Singh Nikam'
   TextField "HmiScreenItemData_6" at 35,192 size 171x28; Text 'Description:'
   TextField "HmiScreenItemData_7" at 241,192 size 524x28; Text '(not configured)'
   Button "Back" at 1,52 size 159x47; TextOff 'Back'
      on Release: ActivateScreen("System screens", 0)

screen "User administration" 800x480, template "Template_1"
   on GenerateScreen: SetTag("Tag_ScreenNumber", 7)
   UserView "HmiScreenItemData" at 8,113 size 791x307
   Button "Back" at 1,52 size 159x47; TextOff 'Back'
      on Release: ActivateScreen("System screens", 0)
   Button "HmiScreenItemData_5" at 173,52 size 159x47; TextOn 'Different jobs'; TextOff 'Login'; PictureOn "Navigates to Different jobs for KTP700 Basic+ PN 17.0.0.0"; PictureOff "Navigates to Different jobs for KTP700 Basic+ PN 17.0.0.0"
      on Press: function_a2a04561()
   Button "HmiScreenItemData_6" at 358,52 size 159x47; TextOn 'Different jobs'; TextOff 'Logout'; PictureOn "Navigates to Different jobs for KTP700 Basic+ PN 17.0.0.0"; PictureOff "Navigates to Different jobs for KTP700 Basic+ PN 17.0.0.0"
      on Press: function_f23ef4c9()

screen "System information" 800x480, template "Template_1"
   on GenerateScreen: SetTag("Tag_ScreenNumber", 8)
   TextField "HmiScreenItemData" at 35,102 size 171x28; Text 'HMI device type:'
   TextField "HmiScreenItemData_1" at 241,102 size 524x28; Text 'KTP700 Basic+ PN 17.0.0.0'
   TextField "HmiScreenItemData_2" at 35,132 size 171x28; Text 'Connection:'
   TextField "HmiScreenItemData_3" at 241,132 size 524x28; Text 'PROFINET (X1)'
   TextField "HmiScreenItemData_4" at 35,162 size 171x28; Text 'PLC:'
   TextField "HmiScreenItemData_5" at 241,162 size 524x28; Text 'SIMATIC S7 1200'
   Button "Back" at 1,52 size 159x47; TextOff 'Back'
      on Release: ActivateScreen("System screens", 0)

screen "Different jobs" 800x480, template "Template_1"
   on GenerateScreen: SetTag("Tag_ScreenNumber", 9)
   Button "Online" at 36,146 size 159x47; TextOff 'Online'
      on Release: function_bb44b551(0)
   Button "Offline" at 36,205 size 159x47; TextOff 'Offline'
      on Release: function_bb44b551(1)
   Button "Transfer" at 36,264 size 159x47; TextOff 'Transfer'
      on Release: function_bb44b551(2)
   Button "Toggle language" at 36,323 size 159x47; TextOff 'Toggle language'
      on Release: function_fb9197e8(-1)
   Button "Stop Runtime" at 207,146 size 159x47; TextOff 'Stop Runtime'
      on Release: StopRuntime(0)
   Button "Back" at 1,52 size 159x47; TextOff 'Back'
      on Release: ActivateScreen("System screens", 0)
*)